TYPE BaudRate EXTENDS SubIndexModuleBase :
STRUCT
END_STRUCT
END_TYPE

(* stored: Version 1.1.0.1, ProductVersion 3.1.4024.3
   DUT BaudRate: Id {5828b878-9918-465a-8d61-ca0192d6244b} *)
